Staubli VAL3: RESET.pgx

public program Reset()
begin

  // This program set the default value of the variables

  // used in the librairy

  //

  //***********************************

  //*****   Conveyor locations    *****

  //***********************************

  //--- Upstream end of the tracking window

  pWinUp[0].trsf={0,0,0,0,0,0}

  pWinUp[1].trsf={0,0,0,0,0,0}

  //

  //--- Donwstream End of the tracking Window

  pWinDown[0].trsf={0,0,0,0,0,0}

  pWinDown[1].trsf={0,0,0,0,0,0}

  //

  //*****************************

  //*****     Numerics      *****

  //*****************************

  //---

  //--- Distance for sync/desync criteria

  nSyncDist=0

end
